(* IEC 61131-3 sources: Takt/book/src/18-showcase/generated/st, 1 file *)

(* ---- lift.st ---- *)
(*
 * Generated by the Takt compiler (taktc). Target: Structured Text (IEC 61131-3).
 * Do not edit by hand: this file is overwritten on every generation.
 * Takt language version 0.19.0.
 *)

(*
 * Такт - шаг логики, не единица времени или расстояния. Положение кабины даёт
 * датчик at_floor (шахтная система позиционирования); движение создаёт привод,
 * а фиксирует - датчик. Выдержка дверей - это отрезок времени, поэтому её порог
 * задан в тактах и подстраивается под частоту устройства.
 *)
FUNCTION_BLOCK Lift
VAR_INPUT
    at_floor : USINT;
    call : USINT;
END_VAR
VAR_OUTPUT
    is_done : BOOL;
    brake : BOOL;
    display : USINT;
    doors_open : BOOL;
    motor_down : BOOL;
    motor_up : BOOL;
END_VAR
VAR
    state : USINT := 0;
    doors : BOOL := FALSE;
    dwell : USINT := 0;
    moving : BOOL := FALSE;
END_VAR
VAR CONSTANT
    DWELL_TICKS : USINT := 3;
END_VAR
    IF state = 0 THEN (* первый скан *)
        moving := FALSE;
        motor_up := FALSE;
        motor_down := FALSE;
        brake := TRUE;
        doors := FALSE;
        doors_open := FALSE;
        state := 6; (* Waiting *)
    END_IF;
    CASE state OF
        1: (* Boarding *)
            dwell := dwell + 1; (* (6) отсчёт ВРЕМЕНИ выдержки (в тактах) *)
            IF dwell >= DWELL_TICKS THEN
                doors := FALSE;
                doors_open := FALSE;
                state := 4; (* Leaving *)
            END_IF;
        2: (* GoingDown *)
            display := at_floor;
            IF at_floor <= call THEN
                moving := FALSE;
                motor_up := FALSE;
                motor_down := FALSE;
                brake := TRUE;
                state := 5; (* Stopping *)
            END_IF;
        3: (* GoingUp *)
            display := at_floor; (* (3) едем; положение — с датчика *)
            IF at_floor >= call THEN
                moving := FALSE;
                motor_up := FALSE;
                motor_down := FALSE;
                brake := TRUE;
                state := 5; (* Stopping *)
            END_IF;
        4: (* Leaving *)
            moving := FALSE;
            motor_up := FALSE;
            motor_down := FALSE;
            brake := TRUE;
            doors := FALSE;
            doors_open := FALSE;
            state := 6; (* Waiting *)
        5: (* Stopping *)
            doors := TRUE;
            doors_open := TRUE;
            dwell := 0;
            state := 1; (* Boarding *)
        6: (* Waiting *)
            display := at_floor; (* (3) индикатор следует за датчиком *)
            IF call = at_floor THEN
                doors := TRUE;
                doors_open := TRUE;
                dwell := 0;
                state := 1; (* Boarding *)
            ELSIF call > at_floor THEN
                moving := TRUE;
                brake := FALSE;
                motor_up := TRUE;
                state := 3; (* GoingUp *)
            ELSIF (call > 0) AND (call < at_floor) THEN
                moving := TRUE;
                brake := FALSE;
                motor_down := TRUE;
                state := 2; (* GoingDown *)
            END_IF;
        7: (* END *)
            state := 7;
    END_CASE;
    is_done := state = 7;
END_FUNCTION_BLOCK
